FUNCTION_BLOCK FB_cycleOutputHZ
VAR
	// last value
	m_Ton : FB_TON;
	m_Time : LREAL;
	m_bEnable :BOOL;
END_VAR

METHOD run : BOOL
VAR_INPUT
	bEnable : BOOL;
	input :LREAL;
END_VAR
m_bEnable:=bEnable;
IF bEnable AND input>0 THEN
	m_Time := 1.0/input;
	m_Ton(IN:= bEnable, PT:= LREAL_TO_TIME(m_Time*1000), Q=> , ET=> );
	IF m_Ton.Q THEN
		m_Ton.reset();
		run := TRUE;
	END_IF
END_IF
END_METHOD

END_FUNCTION_BLOCK

(* stored: Version 1.1.0.1, ProductVersion 3.1.4024.11
   POU FB_cycleOutputHZ: Id {e2d7720e-b6bd-4f29-af28-6199418cfecc}, SpecialFunc None
   Method run: Id {905a3f5d-1781-45d0-9242-f6dfaf4fb169} *)
